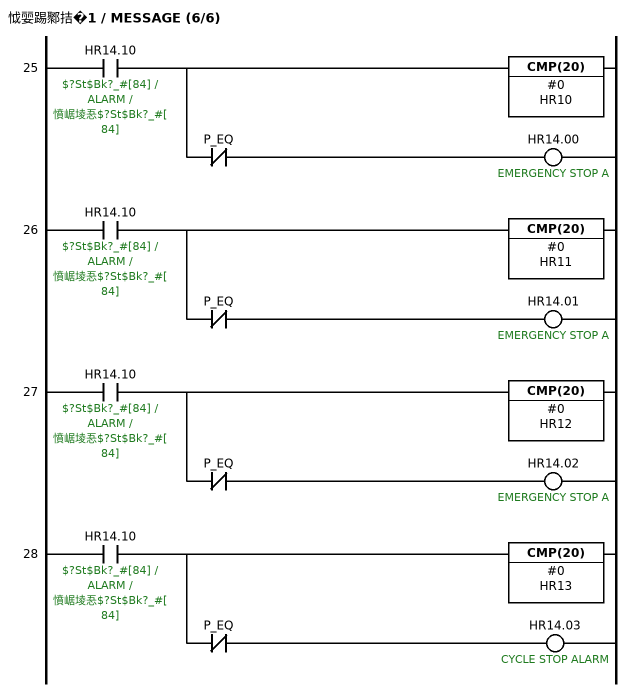
; [picture p24: 怴婯踢鄹拮�1 / MESSAGE, rungs 25-28]
; rung 25
LD HR14.10  ; $?St$Bk?_#[84] / ALARM / 憤崌堎忢$?St$Bk?_#[84]
CMP(20) #0 HR10
ANDNOT P_EQ
OUT HR14.00  ; EMERGENCY STOP A
; rung 26
LD HR14.10  ; $?St$Bk?_#[84] / ALARM / 憤崌堎忢$?St$Bk?_#[84]
CMP(20) #0 HR11
ANDNOT P_EQ
OUT HR14.01  ; EMERGENCY STOP A
; rung 27
LD HR14.10  ; $?St$Bk?_#[84] / ALARM / 憤崌堎忢$?St$Bk?_#[84]
CMP(20) #0 HR12
ANDNOT P_EQ
OUT HR14.02  ; EMERGENCY STOP A
; rung 28
LD HR14.10  ; $?St$Bk?_#[84] / ALARM / 憤崌堎忢$?St$Bk?_#[84]
CMP(20) #0 HR13
ANDNOT P_EQ
OUT HR14.03  ; CYCLE STOP ALARM

### Section DISPLAY

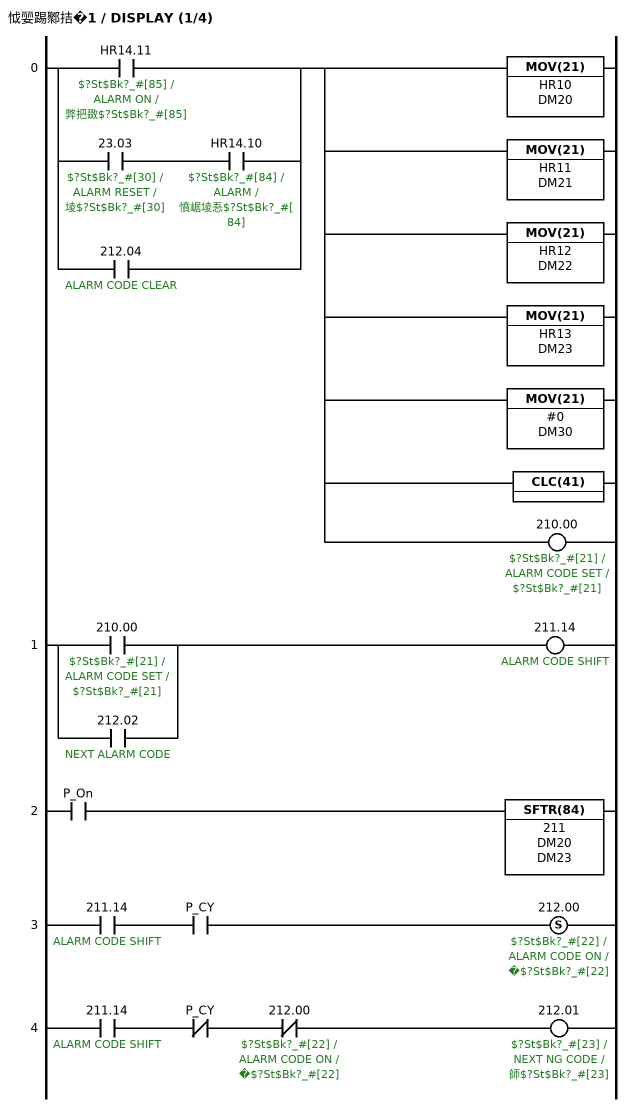
; rung 0
LD HR14.11  ; $?St$Bk?_#[85] / ALARM ON / 弊把敪$?St$Bk?_#[85]
LD 23.03  ; $?St$Bk?_#[30] / ALARM RESET / 堎$?St$Bk?_#[30]
AND HR14.10  ; $?St$Bk?_#[84] / ALARM / 憤崌堎忢$?St$Bk?_#[84]
ORLD
OR 212.04  ; ALARM CODE CLEAR
MOV(21) HR10 DM20
MOV(21) HR11 DM21
MOV(21) HR12 DM22
MOV(21) HR13 DM23
MOV(21) #0 DM30
CLC(41)
OUT 210.00  ; $?St$Bk?_#[21] / ALARM CODE SET / $?St$Bk?_#[21]
; rung 1
LD 210.00  ; $?St$Bk?_#[21] / ALARM CODE SET / $?St$Bk?_#[21]
OR 212.02  ; NEXT ALARM CODE
OUT 211.14  ; ALARM CODE SHIFT
; rung 2
LD P_On
SFTR(84) 211 DM20 DM23
; rung 3
LD 211.14  ; ALARM CODE SHIFT
AND P_CY
SET 212.00  ; $?St$Bk?_#[22] / ALARM CODE ON / �$?St$Bk?_#[22]
; rung 4
LD 211.14  ; ALARM CODE SHIFT
ANDNOT P_CY
ANDNOT 212.00  ; $?St$Bk?_#[22] / ALARM CODE ON / �$?St$Bk?_#[22]
OUT 212.01  ; $?St$Bk?_#[23] / NEXT NG CODE / 師$?St$Bk?_#[23]

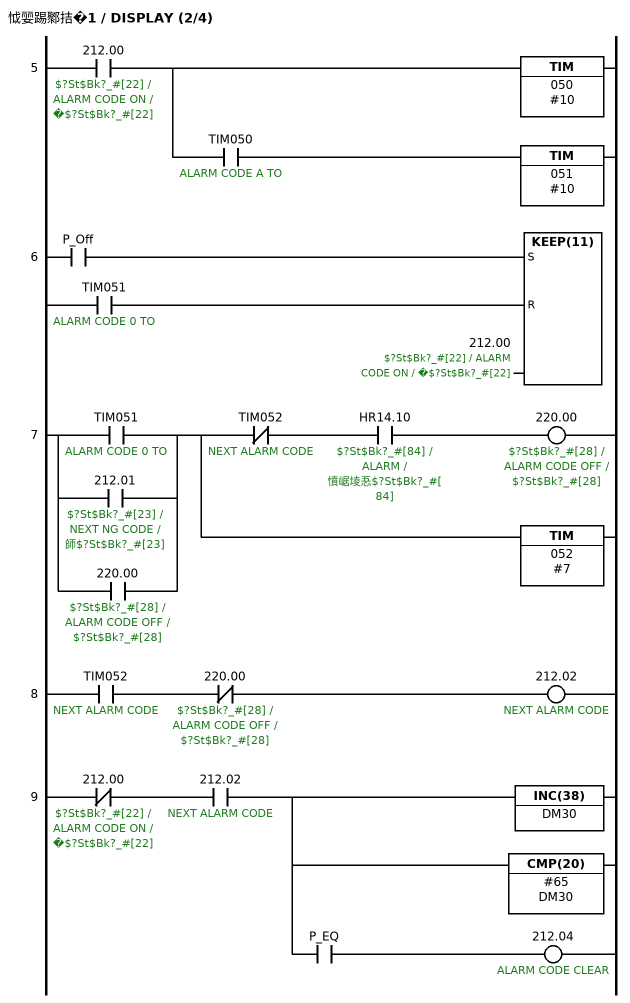
; rung 5
LD 212.00  ; $?St$Bk?_#[22] / ALARM CODE ON / �$?St$Bk?_#[22]
TIM 050 #10
AND TIM050  ; ALARM CODE A TO
TIM 051 #10
; rung 6
LD P_Off
LD TIM051  ; ALARM CODE 0 TO
KEEP(11) 212.00  ; $?St$Bk?_#[22] / ALARM CODE ON / �$?St$Bk?_#[22]
; rung 7
LD TIM051  ; ALARM CODE 0 TO
OR 212.01  ; $?St$Bk?_#[23] / NEXT NG CODE / 師$?St$Bk?_#[23]
OR 220.00  ; $?St$Bk?_#[28] / ALARM CODE OFF / $?St$Bk?_#[28]
OUT TR0
ANDNOT TIM052  ; NEXT ALARM CODE
AND HR14.10  ; $?St$Bk?_#[84] / ALARM / 憤崌堎忢$?St$Bk?_#[84]
OUT 220.00  ; $?St$Bk?_#[28] / ALARM CODE OFF / $?St$Bk?_#[28]
LD TR0
TIM 052 #7
; rung 8
LD TIM052  ; NEXT ALARM CODE
ANDNOT 220.00  ; $?St$Bk?_#[28] / ALARM CODE OFF / $?St$Bk?_#[28]
OUT 212.02  ; NEXT ALARM CODE
; rung 9
LDNOT 212.00  ; $?St$Bk?_#[22] / ALARM CODE ON / �$?St$Bk?_#[22]
AND 212.02  ; NEXT ALARM CODE
INC(38) DM30
CMP(20) #65 DM30
AND P_EQ
OUT 212.04  ; ALARM CODE CLEAR

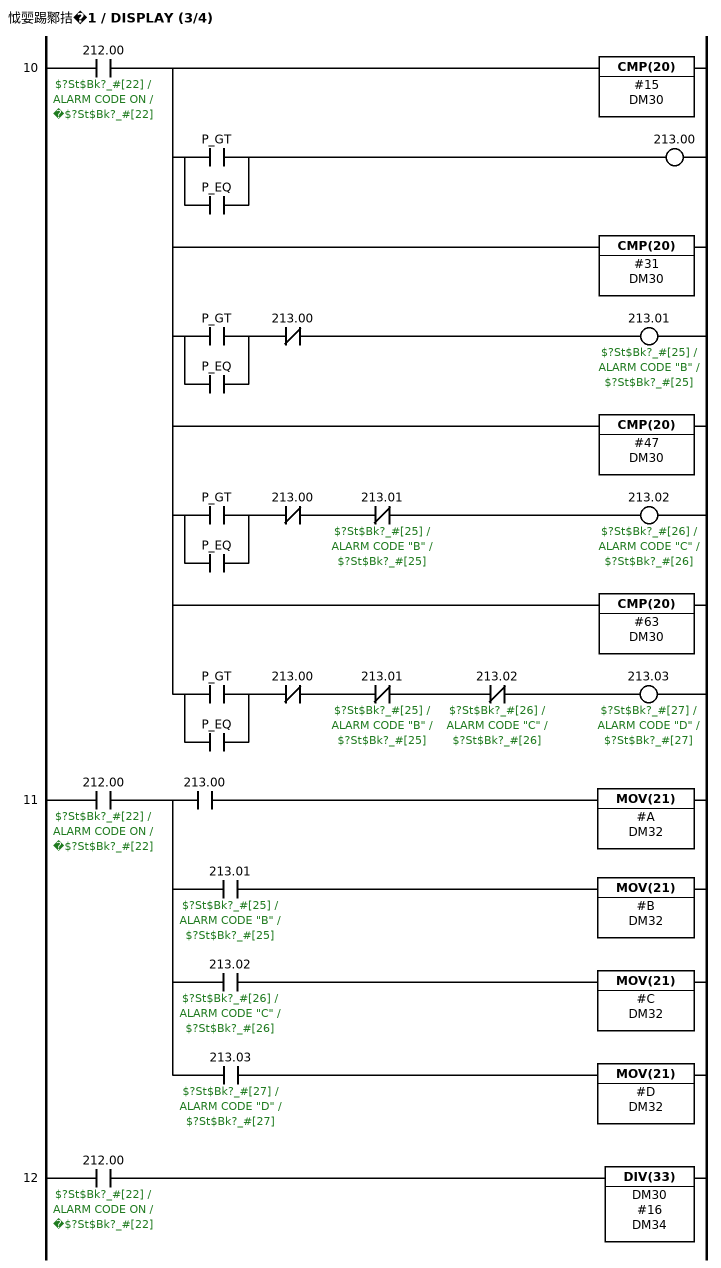
; rung 10
LD 212.00  ; $?St$Bk?_#[22] / ALARM CODE ON / �$?St$Bk?_#[22]
OUT TR0
CMP(20) #15 DM30
LD P_GT
OR P_EQ
ANDLD
OUT 213.00
LD TR0
CMP(20) #31 DM30
LD P_GT
OR P_EQ
ANDLD
ANDNOT 213.00
OUT 213.01  ; $?St$Bk?_#[25] / ALARM CODE "B" / $?St$Bk?_#[25]
LD TR0
CMP(20) #47 DM30
LD P_GT
OR P_EQ
ANDLD
ANDNOT 213.00
ANDNOT 213.01  ; $?St$Bk?_#[25] / ALARM CODE "B" / $?St$Bk?_#[25]
OUT 213.02  ; $?St$Bk?_#[26] / ALARM CODE "C" / $?St$Bk?_#[26]
LD TR0
CMP(20) #63 DM30
LD P_GT
OR P_EQ
ANDLD
ANDNOT 213.00
ANDNOT 213.01  ; $?St$Bk?_#[25] / ALARM CODE "B" / $?St$Bk?_#[25]
ANDNOT 213.02  ; $?St$Bk?_#[26] / ALARM CODE "C" / $?St$Bk?_#[26]
OUT 213.03  ; $?St$Bk?_#[27] / ALARM CODE "D" / $?St$Bk?_#[27]
; rung 11
LD 212.00  ; $?St$Bk?_#[22] / ALARM CODE ON / �$?St$Bk?_#[22]
OUT TR0
AND 213.00
MOV(21) #A DM32
LD TR0
AND 213.01  ; $?St$Bk?_#[25] / ALARM CODE "B" / $?St$Bk?_#[25]
MOV(21) #B DM32
LD TR0
AND 213.02  ; $?St$Bk?_#[26] / ALARM CODE "C" / $?St$Bk?_#[26]
MOV(21) #C DM32
LD TR0
AND 213.03  ; $?St$Bk?_#[27] / ALARM CODE "D" / $?St$Bk?_#[27]
MOV(21) #D DM32
; rung 12
LD 212.00  ; $?St$Bk?_#[22] / ALARM CODE ON / �$?St$Bk?_#[22]
DIV(33) DM30 #16 DM34

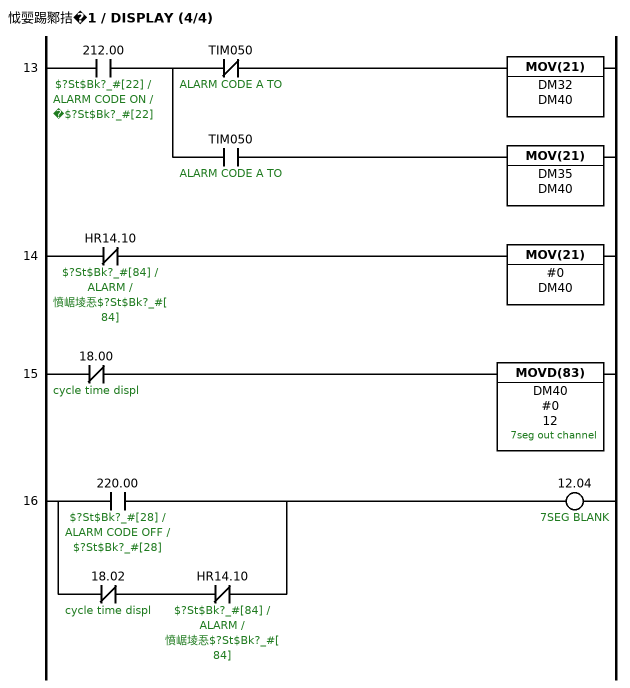
; rung 13
LD 212.00  ; $?St$Bk?_#[22] / ALARM CODE ON / �$?St$Bk?_#[22]
OUT TR0
ANDNOT TIM050  ; ALARM CODE A TO
MOV(21) DM32 DM40
LD TR0
AND TIM050  ; ALARM CODE A TO
MOV(21) DM35 DM40
; rung 14
LDNOT HR14.10  ; $?St$Bk?_#[84] / ALARM / 憤崌堎忢$?St$Bk?_#[84]
MOV(21) #0 DM40
; rung 15
LDNOT 18.00  ; cycle time displ
MOVD(83) DM40 #0 12  ; 7seg out channel
; rung 16
LD 220.00  ; $?St$Bk?_#[28] / ALARM CODE OFF / $?St$Bk?_#[28]
LDNOT 18.02  ; cycle time displ
ANDNOT HR14.10  ; $?St$Bk?_#[84] / ALARM / 憤崌堎忢$?St$Bk?_#[84]
ORLD
OUT 12.04  ; 7SEG BLANK

### Section END
; rung 0
END(01)